Omron CX-Programmer project NuevoProyecto (CX-Programmer 9.61)

# PLC Caramelos: CJ2M CPU31
I/O table (CPU CJ2M-CPU31): rack 0 slot 11 CJ2M-EIP21

## Program NuevoPrograma1 (cyclic task 0)
Local symbols
CarameloA 0.02 BOOL
CarameloB 0.03 BOOL
CincoCents 0.00 BOOL
Devolviendo 1.10 BOOL
DiezCents 0.01 BOOL
Extraer 0.04 BOOL
ExtrayendoA 1.08 BOOL
ExtrayendoB 1.09 BOOL
LedCinco 1.05 BOOL
LedCuatro 1.04 BOOL
LedDos 1.02 BOOL
LedReady 1.00 BOOL
LedTres 1.03 BOOL
LedUno 1.01 BOOL
ListoA 1.06 BOOL
ListoB 1.07 BOOL
P0 2.00 BOOL
P1 2.01 BOOL
P2 2.02 BOOL
P3 2.03 BOOL
P4 2.04 BOOL
P5 2.05 BOOL
P6 2.06 BOOL
P7 2.07 BOOL
P8 2.08 BOOL

### Section Sección1

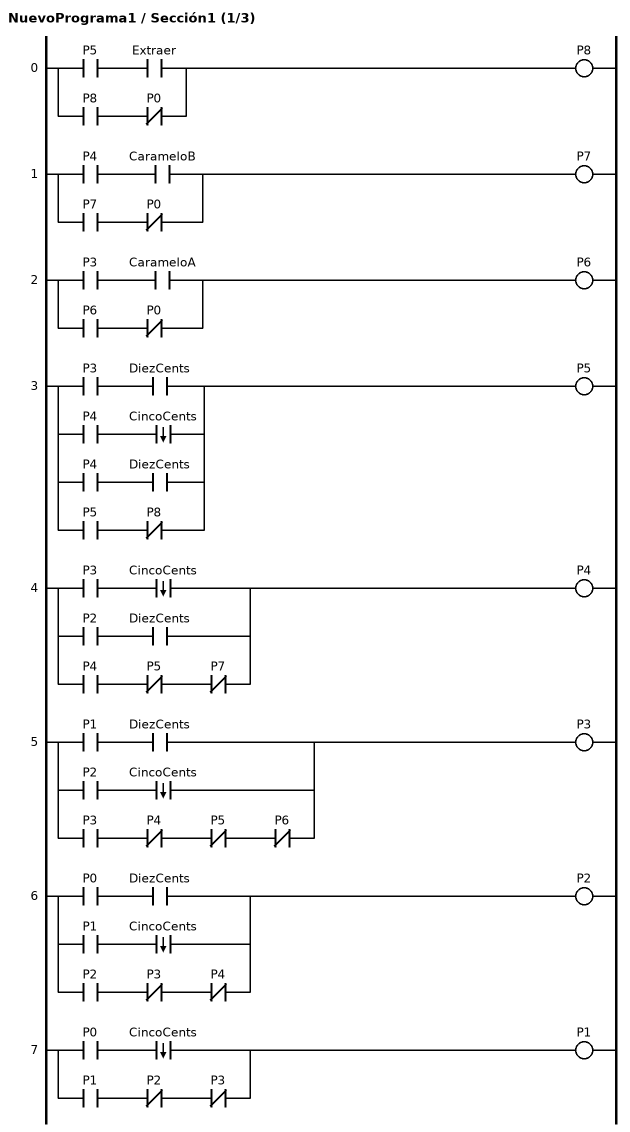
; rung 0
LD P5
AND Extraer
LD P8
ANDNOT P0
ORLD
OUT P8
; rung 1
LD P4
AND CarameloB
LD P7
ANDNOT P0
ORLD
OUT P7
; rung 2
LD P3
AND CarameloA
LD P6
ANDNOT P0
ORLD
OUT P6
; rung 3
LD P3
AND DiezCents
LD P4
%AND CincoCents
ORLD
LD P4
AND DiezCents
ORLD
LD P5
ANDNOT P8
ORLD
OUT P5
; rung 4
LD P3
%AND CincoCents
LD P2
AND DiezCents
ORLD
LD P4
ANDNOT P5
ANDNOT P7
ORLD
OUT P4
; rung 5
LD P1
AND DiezCents
LD P2
%AND CincoCents
ORLD
LD P3
ANDNOT P4
ANDNOT P5
ANDNOT P6
ORLD
OUT P3
; rung 6
LD P0
AND DiezCents
LD P1
%AND CincoCents
ORLD
LD P2
ANDNOT P3
ANDNOT P4
ORLD
OUT P2
; rung 7
LD P0
%AND CincoCents
LD P1
ANDNOT P2
ANDNOT P3
ORLD
OUT P1

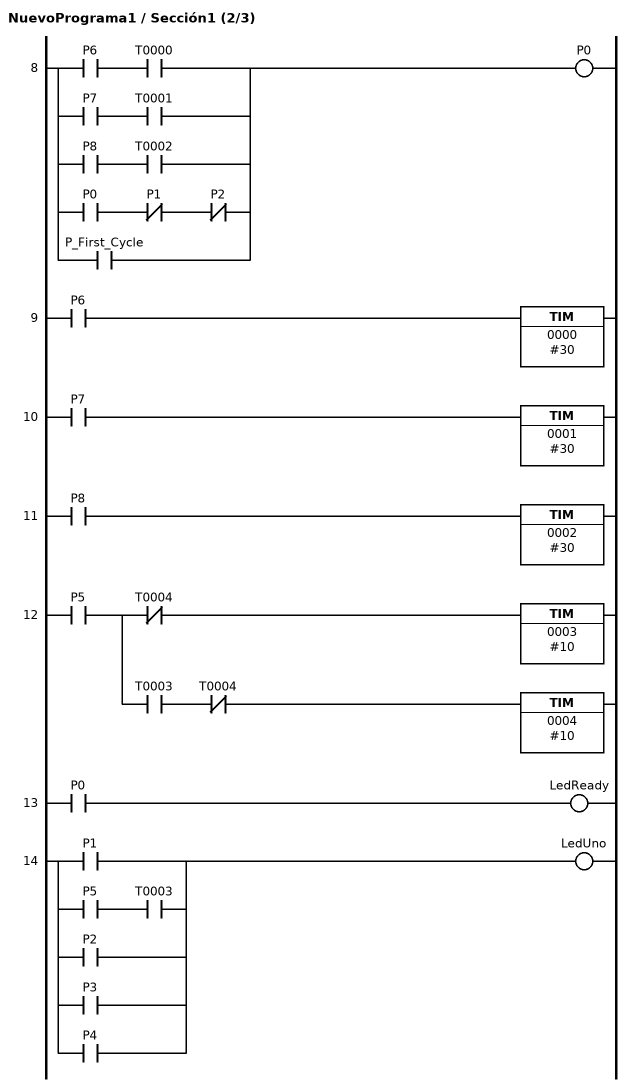
; rung 8
LD P6
AND T0000
LD P7
AND T0001
ORLD
LD P8
AND T0002
ORLD
LD P0
ANDNOT P1
ANDNOT P2
ORLD
OR P_First_Cycle
OUT P0
; rung 9
LD P6
TIM 0000 #30
; rung 10
LD P7
TIM 0001 #30
; rung 11
LD P8
TIM 0002 #30
; rung 12
LD P5
OUT TR0
ANDNOT T0004
TIM 0003 #10
LD TR0
AND T0003
ANDNOT T0004
TIM 0004 #10
; rung 13
LD P0
OUT LedReady
; rung 14
LD P1
LD P5
AND T0003
ORLD
OR P2
OR P3
OR P4
OUT LedUno

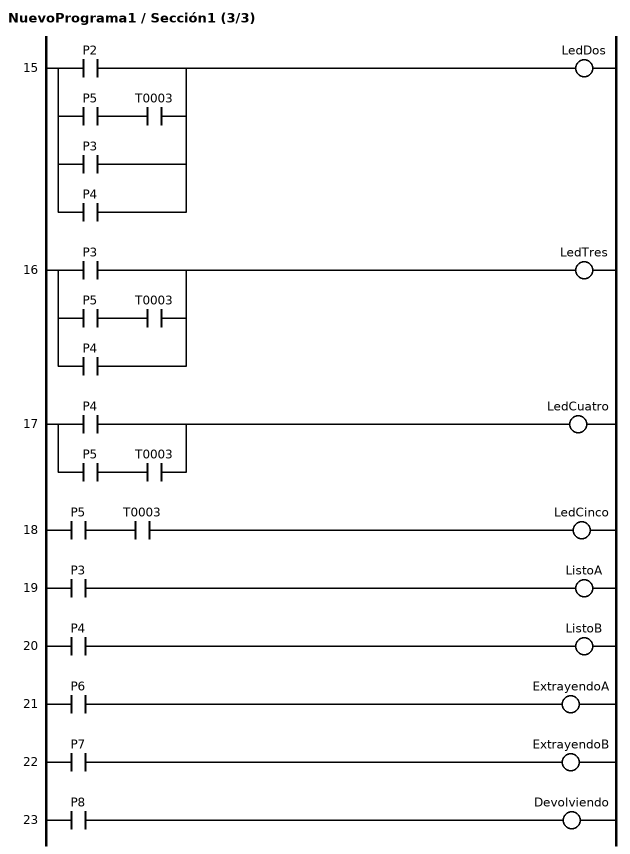
; rung 15
LD P2
LD P5
AND T0003
ORLD
OR P3
OR P4
OUT LedDos
; rung 16
LD P3
LD P5
AND T0003
ORLD
OR P4
OUT LedTres
; rung 17
LD P4
LD P5
AND T0003
ORLD
OUT LedCuatro
; rung 18
LD P5
AND T0003
OUT LedCinco
; rung 19
LD P3
OUT ListoA
; rung 20
LD P4
OUT ListoB
; rung 21
LD P6
OUT ExtrayendoA
; rung 22
LD P7
OUT ExtrayendoB
; rung 23
LD P8
OUT Devolviendo

### Section END
; rung 0
END(001)